(* LS Electric XG5000 project: Perform Liquid Level Control *)
(* PLC LSPLC *)
(* module base 0 slot 0: Input/Output Module:XEC-DR32H (DC 24V input 16 points, relay output 16 points) *)
(* module base 0 slot 1: Analog IO Module:XBF-AH04A (A/D Voltage/Current 2 Ch, D/A Voltage/Current 2 Ch) *)
VAR_GLOBAL
    OUT : SINT;
    OUT_PUT : WORD;
    _01_AD01_DATA_ARY AT %UW0.1.4 : ARRAY[0..1] OF WORD; (* Analog IO Module: Input each CH Data *)
END_VAR

PROGRAM NewProgram (* task: Scan Program *)
VAR
    on_off : BOOL;
    pump AT %QX0.0.1 : BOOL;
    start_switch AT %IX0.0.1 : BOOL;
    stop_switch AT %IX0.0.2 : BOOL;
    sys1_on : BOOL;
    sys_off : BOOL;
    sys_on AT %QX0.0.2 : BOOL;
END_VAR
VAR_EXTERNAL
    OUT : SINT;
    OUT_PUT : WORD;
    _01_AD01_DATA_ARY : ARRAY[0..1] OF WORD; (* AT %UW0.1.4 *) (* Analog IO Module: Input each CH Data *)
END_VAR
VAR
    _p1 : BOOL;
END_VAR

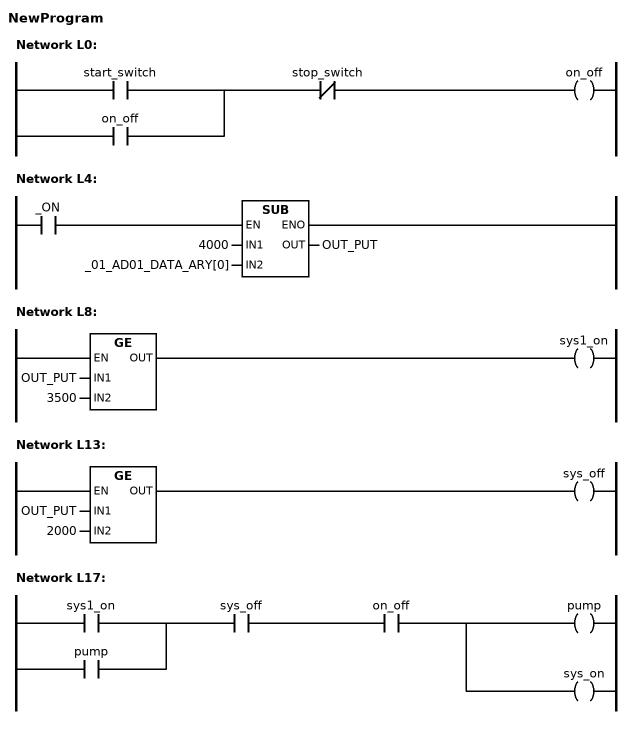
(* Rung L0 *)
on_off := (start_switch OR on_off) AND NOT stop_switch;
(* Rung L4 *)
IF _ON THEN OUT_PUT := 4000 - _01_AD01_DATA_ARY[0]; END_IF;
(* Rung L8 *)
sys1_on := OUT_PUT >= 3500;
(* Rung L13 *)
sys_off := OUT_PUT >= 2000;
(* Rung L17 *)
_p1 := (sys1_on OR pump) AND sys_off AND on_off;
pump := _p1;
sys_on := _p1;
END_PROGRAM